// Mitsubishi GX Works2 project: 주석 작성   PLC: Q03UDV

PROGRAM MAIN
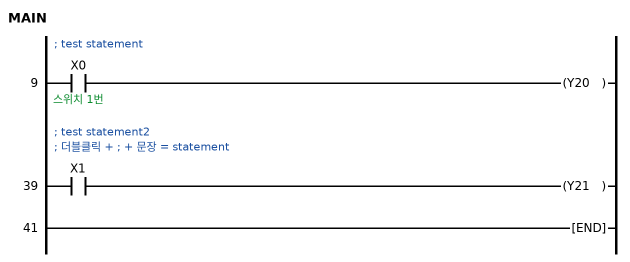
; test statement
9     LD      X0  ; 스위치 1번
      OUT     Y20
; test statement2
; 더블클릭 + ; + 문장 = statement
39    LD      X1
      OUT     Y21
41    END
END_PROGRAM
